///Checks if the returned HRESULT is success
FUNCTION Success : BOOL
VAR_INPUT
    hr : HRESULT;
END_VAR
VAR
END_VAR

Success := (hr >= 0);

END_FUNCTION

(* stored: Version 1.1.0.1, ProductVersion 3.1.4020.12
   POU Success: Id {1f2321bb-8405-4e96-a878-5b581c40e42d}, SpecialFunc None *)
